PROGRAM PhysicalSystemTest
VAR
	ABB: INT;
	TwoSecTimer: TON;
	mxTimerStart:BOOL;
	mxTimerDone:BOOL;
END_VAR

CASE ABB OF
	0:
		IF CommData.qxPLCStrobe THEN
			ABB:=10;
		END_IF
	10:
		IF CommData.qwOrderRobot > 0 THEN
			CommData.iwReplyRobot:=CommData.qwOrderRobot+1;
			mxTimerStart:=TRUE;
			ABB:=20;
		END_IF
	20:
		IF mxTimerDone THEN
			CommData.ixRobotStrobe :=TRUE;
			mxTimerStart:=FALSE;
			ABB:=30;
		END_IF
	30:
		IF NOT CommData.qxPLCStrobe THEN
			mxTimerStart:=TRUE;
			ABB:=40;
		END_IF
	40:
		IF mxTimerDone THEN
			CommData.iwReplyRobot:=0;
			CommData.ixRobotStrobe :=FALSE;
			mxTimerStart:=FALSE;
			ABB:=50;
		END_IF
	50:
		mxTimerStart:=TRUE;
		IF mxTimerDone THEN
			mxTimerStart:=FALSE;
			CommData.iwProgressRobot:=90;
			ABB:=60;
		END_IF
	60:
		CommData.ixRobotStrobe :=TRUE;
		mxTimerStart:=TRUE;
		ABB:=70;
	70:
		IF mxTimerDone AND CommData.qxPLCStrobe THEN
			mxTimerStart:=FALSE;
			CommData.iwProgressRobot:=0;
			ABB:=80;
		END_IF
	80:
		mxTimerStart:=TRUE;
		IF mxTimerDone THEN
			mxTimerStart:=FALSE;
			CommData.ixRobotStrobe :=FALSE;
			ABB:=90;
		END_IF
	90:
		IF NOT CommData.qxPLCStrobe THEN
			ABB:=0;
		END_IF
END_CASE



TwoSecTimer(IN:= mxTimerStart, PT:= T#2S, Q=> mxTimerDone, ET=> );

END_PROGRAM

(* stored: Version 1.1.0.1, ProductVersion 3.1.4024.10
   POU PhysicalSystemTest: Id {18e66b61-bfa1-469f-ba97-fead9c46c956}, SpecialFunc None *)
